{attribute 'GeneratedUsingTerminal: KL9900-0064'}
{attribute addProperty BoxType "KL9900-0064"}
{attribute addProperty Id "Key_1AT %I*BOOL0Key_2AT %I*BOOL0Key_3AT %I*BOOL0Key_4AT %I*BOOL0Input_1AT %I*BOOL0Input_2AT %I*BOOL0Input_3AT %I*BOOL0Input_4AT %I*BOOL0LED_1AT %Q*BOOL0LED_2AT %Q*BOOL0LED_3AT %Q*BOOL0LED_4AT %Q*BOOL0"}
{attribute addProperty CRC "252500288"}
{attribute addProperty Size "0"}
TYPE Channel_0F0CD940 :
STRUCT
	{attribute addProperty Name "Key_1"}
	Key_1 AT %I* : BOOL;
	{attribute addProperty Name "Key_2"}
	Key_2 AT %I* : BOOL;
	{attribute addProperty Name "Key_3"}
	Key_3 AT %I* : BOOL;
	{attribute addProperty Name "Key_4"}
	Key_4 AT %I* : BOOL;
	{attribute addProperty Name "Input_1"}
	Input_1 AT %I* : BOOL;
	{attribute addProperty Name "Input_2"}
	Input_2 AT %I* : BOOL;
	{attribute addProperty Name "Input_3"}
	Input_3 AT %I* : BOOL;
	{attribute addProperty Name "Input_4"}
	Input_4 AT %I* : BOOL;
	{attribute addProperty Name "LED_1"}
	LED_1 AT %Q* : BOOL;
	{attribute addProperty Name "LED_2"}
	LED_2 AT %Q* : BOOL;
	{attribute addProperty Name "LED_3"}
	LED_3 AT %Q* : BOOL;
	{attribute addProperty Name "LED_4"}
	LED_4 AT %Q* : BOOL;
END_STRUCT
END_TYPE

(* stored: Version 1.2.0.0, ProductVersion 3.1.4024.9
   DUT Channel_0F0CD940: Id {80637602-ca55-48ae-b70d-b8de5884c53e} *)
